{attribute 'qualified_only'}
{attribute 'strict'}
{attribute 'to_string'}
TYPE
    E_TaskState : (
        IDLE,
        PENDING,
        ACTIVE,
        MANUAL,
        COMPLETE,
        ERROR,
        RECOVERY,
        ABORT,
        ABORT_RETRY,
        INVALID
    );
END_TYPE

(* stored: Version 1.1.0.1
   DUT E_TaskState: Id {68f654e0-dbba-4b08-960f-359f61506ae1} *)
